TYPE T_Ctrl_SIf_MOD_In :
STRUCT	
	// Inputs from global module for general supervision 
	// Emergency circuit ok
	bolEmergencyOffOk: T_Ctrl_IoBool;
	// No general error active, will be set to FALSE if there is an global error like e.g. over temperature in cabinet. 
	bolNoGeneralError: T_Ctrl_IoBool;
END_STRUCT
END_TYPE

(* stored: Version 1.1.0.1, ProductVersion 3.1.0.19
   DUT T_Ctrl_SIf_MOD_In: Id {c935e795-2dfd-4a28-8708-5ac7a294862e} *)
